VISUALIZATION VISU  // 2x2
END_VISUALIZATION

(* stored: Version 1.1.0.1, ProductVersion 3.1.4022.18
   Visu VISU: Id {ff0741aa-bea5-4772-b45e-584e83db76b9} *)
